// TIA Portal V20 export
TYPE "typeCmControlNode"
// stored: Namespace Unit1.Em2
   STRUCT
      Interlock { ExternalWritable := 'False'} : "Unit1.Em2.typeCmControlNodeInterlock";
   END_STRUCT;
END_TYPE
